Staubli VAL3: message.pgx

public program message(string& message[], num index)
// English IF message
begin
  // lenght of message
  //
  switch index
    case 0
      message="Voulez-vous entrer dans le:"
    break
    case 1
      message="< SI ASSISTANT >"
    break
    case 2
      message="Sélect. le type de condition pour vérifier"
    break
    case 3
      message="Sélect. l'Entrée"
    break
    case 4
      message="Sélect. la Sortie"
    break
    case 5
      message="Sélect. L'entrée EMAP"
    break
    case 6
      message="Sélect. la voie comment faire fonctionner l'instruction"
    break
    case 7
      message="Sélect. l'instruction pour associer vers le:"
    break
    case 8
      message="Sélect. de la liste le: "
    break
  endSwitch
end
